// TIA Portal V21 export
VAR_GLOBAL   // PLC tag table "KAllParatia"
END_VAR
VAR_GLOBAL CONSTANT   // user constants
   KAllParatia_OvertimeMovimento : Int := 1;   // Overtime Bewegung / Movement overtime / Overtime movimiento / Overtime mouvement / Overtime movimento
   KAllParatia_TermicoIntervenuto : Int := 2;   // Thermisch Interventioniert / Intervened Thermal / Térmico Intervención / Thermique Intervenu / Termico Intervenuto
   KAllParatia_SezionatoreAperto : Int := 3;   // Trennschalter offen / Disconnector open / Seccionador abierto / Sectionneur ouvert / Sezionatore aperto
END_VAR
